DATA_BLOCK "ST10_Flow11_A2TableScan_iDB"
{ S7_Optimized_Access := 'TRUE' }
VERSION : 0.1
NON_RETAIN
// ATTRIBUTES
// AUTO_NUMBER = False
// BLOCK_NUMBER = 1081
// END_ATTRIBUTES
"ST10_Flow11_A2TableScan"

BEGIN

END_DATA_BLOCK

